SYSTEM A1T1_a (* Simple traffic light *)
  (* Standard: 61499-1 *)
  (* Version 0.1, 2009-03-05, JHC, Holobloc Inc., Deleted Application. *)
  (* Version 0.0, 2004-01-10, JHC, Rockwell Automation, Modified from FLASHERT_TESTD. *)
  DEVICE CTL_PANEL : FRAME_DEVICE(BOUNDS := [50,100,325,100], GRID := [1,1])
    RESOURCE RES1 : PANEL_RESOURCE
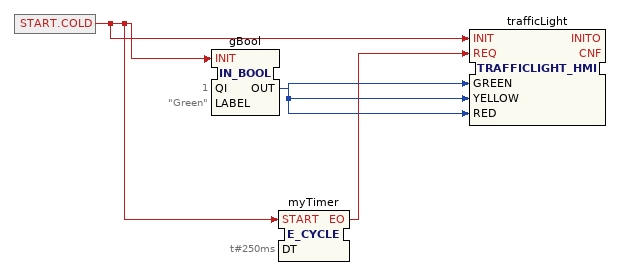
      FBS
        trafficLight : TRAFFICLIGHT_HMI;
        myTimer : E_CYCLE(DT := t#250ms);
        gBool : IN_BOOL(QI := 1, LABEL := "Green");
      END_FBS
      EVENT_CONNECTIONS
        START.COLD TO trafficLight.INIT;
        myTimer.EO TO trafficLight.REQ;
        START.COLD TO myTimer.START;
        START.COLD TO gBool.INIT;
      END_CONNECTIONS
      DATA_CONNECTIONS
        gBool.OUT TO trafficLight.GREEN;
        gBool.OUT TO trafficLight.YELLOW;
        gBool.OUT TO trafficLight.RED;
      END_CONNECTIONS
    END_RESOURCE
  END_DEVICE
END_SYSTEM
